FUNCTION_BLOCK FB_EmagGT
VAR_INPUT
END_VAR
VAR_OUTPUT
END_VAR
VAR
END_VAR

END_FUNCTION_BLOCK

(* stored: Version 1.1.0.1, ProductVersion 3.1.4024.10
   POU FB_EmagGT: Id {4cf53386-82f7-4bad-a149-3dcf35915689}, SpecialFunc None *)
